FUNCTION SclByteDMX : BYTE
VAR_INPUT
	byUnscaled	: BYTE;
END_VAR
VAR
END_VAR

IF byUnscaled = 0 THEN
	SclByteDMX	:= 0;
ELSE
	SclByteDMX	:= 255;
END_IF

END_FUNCTION

(* stored: Version 1.1.0.1, ProductVersion 3.1.4024.6
   POU SclByteDMX: Id {2d2893c9-a97d-46ac-9240-1f212077316c}, SpecialFunc None *)
